TYPE ST_FormingMoldErrors :
STRUCT
	
	Error1: BOOL;

END_STRUCT
END_TYPE

(* stored: Version 1.1.0.1, ProductVersion 3.1.4020.12
   DUT ST_FormingMoldErrors: Id {75341e35-fc3a-460a-bb7b-89602b4ac15d} *)
